// TIA Portal project "TankSimulation.TiaPortalProject" (V14)

(* hardware
DEVICE "S7-1200 station_2"  S7-1200 Station
   slot 0: "Rack_0"  S7-1200 Rack  Rack  V1.0
   slot 1: "TankSimulation"  CPU 1212C DC/DC/Rly  6ES7 212-1HE31-0XB0  V3.0
*)

// ===== PLC "TankSimulation"  CPU 1212C DC/DC/Rly =====

VAR_GLOBAL   // PLC tag table "Default tag table"
   "Tag_1" AT %M10.0 : Bool;
   "System_Byte" AT %MB1 : Byte;
   "FirstScan" AT %M1.0 : Bool;
   "DiagStatusUpdate" AT %M1.1 : Bool;
   "AlwaysTRUE" AT %M1.2 : Bool;
   "AlwaysFALSE" AT %M1.3 : Bool;
   "Clock_Byte" AT %MB0 : Byte;
   "Clock_10Hz" AT %M0.0 : Bool;
   "Clock_5Hz" AT %M0.1 : Bool;
   "Clock_2.5Hz" AT %M0.2 : Bool;
   "Clock_2Hz" AT %M0.3 : Bool;
   "Clock_1.25Hz" AT %M0.4 : Bool;
   "Clock_1Hz" AT %M0.5 : Bool;
   "Clock_0.625Hz" AT %M0.6 : Bool;
   "Clock_0.5Hz" AT %M0.7 : Bool;
END_VAR

DATA_BLOCK "Snap7interfaceDb"   // DB1
{ S7_Optimized_Access := 'FALSE' }
VERSION : 0.1
   VAR
      PumpManual : Bool;
      FlowManual : Bool;
      StartAuto : Bool;
      StopAuto : Bool;
      TankLevel : Real;
      ParameterFlowSpeed : Real := 1.0;
      ParameterPumpSpeed : Real := 2.0;
      AutoState : Bool;
      PumpsState : Bool;
      FlowState : Bool;
      RealFlowSpeed : Real;
      RealPumpSpeed : Real;
   END_VAR
BEGIN
END_DATA_BLOCK

DATA_BLOCK "StateMachineDb"   // DB2
{ S7_Optimized_Access := 'TRUE' }
VERSION : 0.1
// stored: InstanceOfName StateMachine
"StateMachine"
BEGIN
END_DATA_BLOCK

DATA_BLOCK "AlarmsDb"   // DB3
{ S7_Optimized_Access := 'FALSE' }
VERSION : 0.1
   VAR
      GlobalAlarm : Bool;
      PumpSpeedHigh : Bool;
      FlowSpeedHigh : Bool;
   END_VAR
BEGIN
END_DATA_BLOCK

FUNCTION_BLOCK "StateMachine"   // FB1, LAD
{ S7_Optimized_Access := 'TRUE' }
VERSION : 0.1
   VAR
      Clock100ms : Bool;
      "Timer" : IEC_TIMER;
      Test : Bool;
      PumpRunning : Bool;
      AutoRunning : Bool;
      FlowRunning : Bool;
      CurrentState : Byte;
   END_VAR
   VAR_TEMP   // added for the SCL form of the ladder/FBD networks
      _w1 : Bool;
   END_VAR
BEGIN

REGION Network 1: Clock 100ms
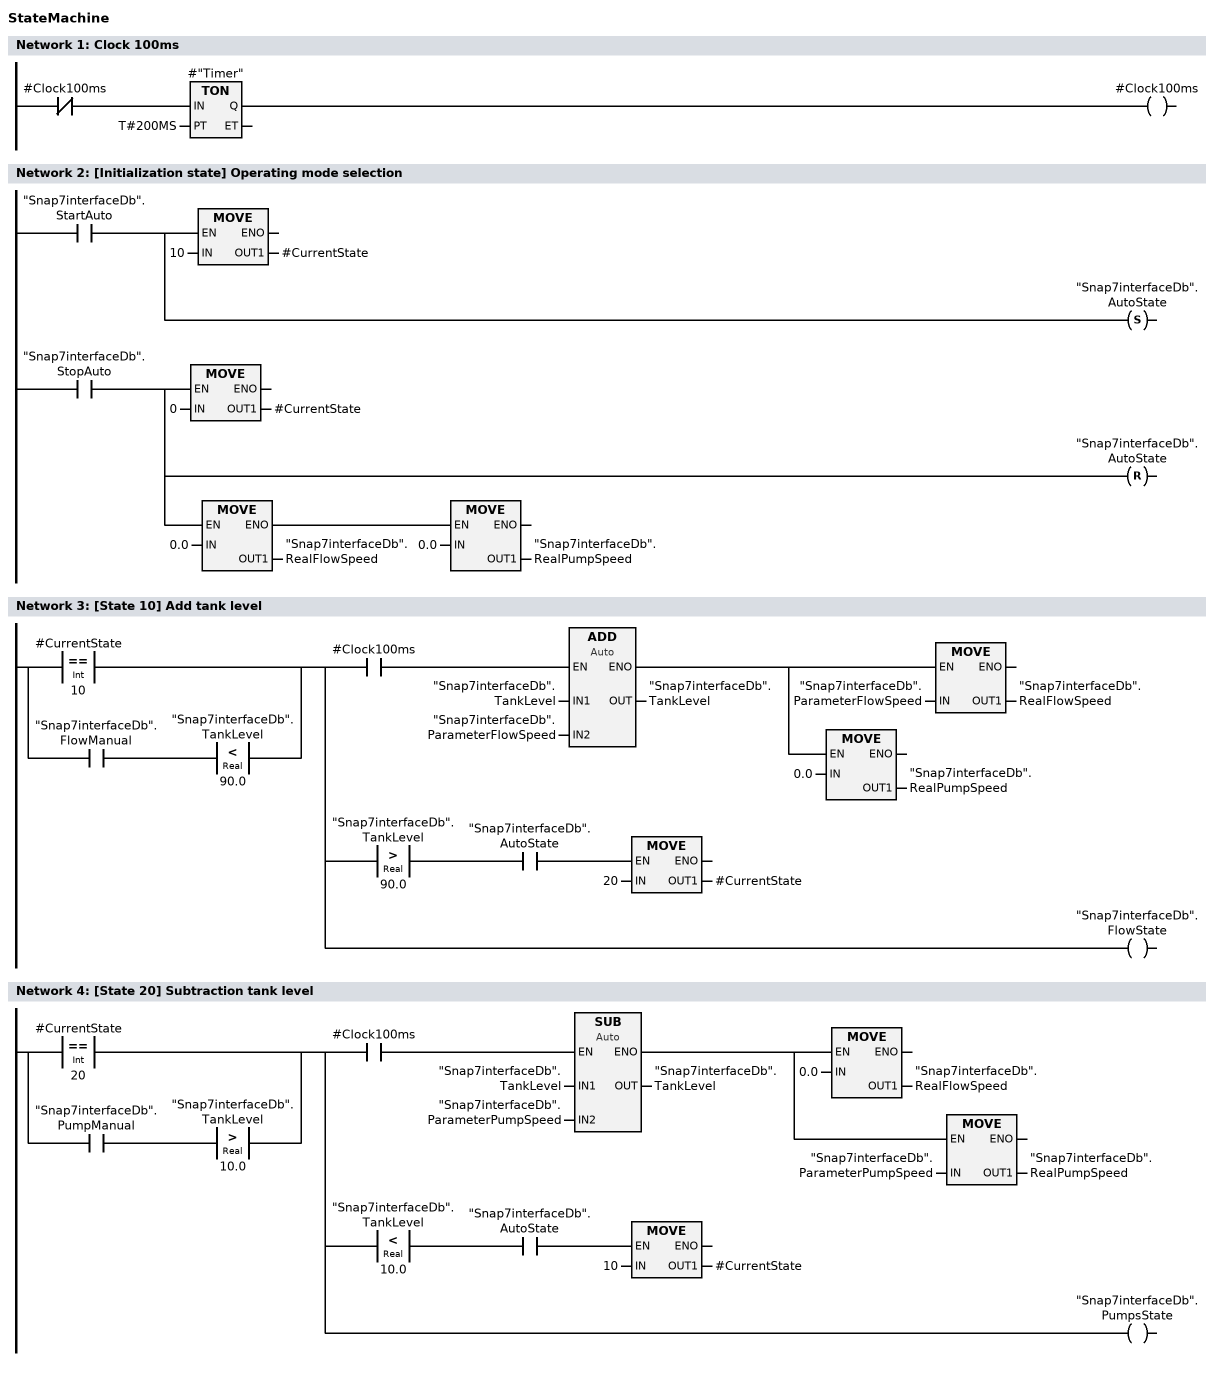
   #"Timer".TON(IN := NOT #Clock100ms, PT := T#200MS);
   #Clock100ms := #"Timer".Q;
END_REGION

REGION Network 2: [Initialization state] Operating mode selection
   RUNG wire#powerrail
      Contact( "Snap7interfaceDb".StartAuto )
      wire#w1
      { S7_GenerateENO := "TRUE" } Move(in := 10, out1 => #CurrentState)
   END_RUNG
   RUNG wire#w1
      S_Coil( "Snap7interfaceDb".AutoState )
   END_RUNG
   RUNG wire#powerrail
      Contact( "Snap7interfaceDb".StopAuto )
      wire#w2
      { S7_GenerateENO := "TRUE" } Move(in := 0, out1 => #CurrentState)
   END_RUNG
   RUNG wire#w2
      R_Coil( "Snap7interfaceDb".AutoState )
   END_RUNG
   RUNG wire#w2
      { S7_GenerateENO := "TRUE" } Move(in := 0.0, out1 => "Snap7interfaceDb".RealFlowSpeed)
      { S7_GenerateENO := "TRUE" } Move(in := 0.0, out1 => "Snap7interfaceDb".RealPumpSpeed)
   END_RUNG
   // the same network as SCL:
   // ENO of a box is taken as its EN; it also drops when the box reports an error
   IF "Snap7interfaceDb".StartAuto THEN
       #CurrentState := 10;
       "Snap7interfaceDb".AutoState := TRUE;
   END_IF;
   IF "Snap7interfaceDb".StopAuto THEN
       #CurrentState := 0;
       "Snap7interfaceDb".AutoState := FALSE;
       "Snap7interfaceDb".RealFlowSpeed := 0.0;
       "Snap7interfaceDb".RealPumpSpeed := 0.0;
   END_IF;
END_REGION

REGION Network 3: [State 10] Add tank level
   RUNG wire#powerrail
      { S7_Templates := "SrcType := Int" } EQ_Contact(in1 := #CurrentState, in2 := 10)
      wire#w1
      Contact( #Clock100ms )
      { S7_GenerateENO := "TRUE" } Add(in1 := "Snap7interfaceDb".TankLevel, in2 := "Snap7interfaceDb".ParameterFlowSpeed, out => "Snap7interfaceDb".TankLevel)
      wire#w2
      { S7_GenerateENO := "TRUE" } Move(in := "Snap7interfaceDb".ParameterFlowSpeed, out1 => "Snap7interfaceDb".RealFlowSpeed)
   END_RUNG
   RUNG wire#powerrail
      Contact( "Snap7interfaceDb".FlowManual )
      { S7_Templates := "SrcType := Real" } LT_Contact(in1 := "Snap7interfaceDb".TankLevel, in2 := 90.0)
   END_RUNG wire#w1
   RUNG wire#w2
      { S7_GenerateENO := "TRUE" } Move(in := 0.0, out1 => "Snap7interfaceDb".RealPumpSpeed)
   END_RUNG
   RUNG wire#w1
      { S7_Templates := "SrcType := Real" } GT_Contact(in1 := "Snap7interfaceDb".TankLevel, in2 := 90.0)
      Contact( "Snap7interfaceDb".AutoState )
      { S7_GenerateENO := "TRUE" } Move(in := 20, out1 => #CurrentState)
   END_RUNG
   RUNG wire#w1
      Coil( "Snap7interfaceDb".FlowState )
   END_RUNG
   // the same network as SCL:
   // ENO of a box is taken as its EN; it also drops when the box reports an error
   #_w1 := (#CurrentState = 10) OR ("Snap7interfaceDb".FlowManual AND ("Snap7interfaceDb".TankLevel < 90.0));
   IF #_w1 AND #Clock100ms THEN
       "Snap7interfaceDb".TankLevel := "Snap7interfaceDb".TankLevel + "Snap7interfaceDb".ParameterFlowSpeed;
       "Snap7interfaceDb".RealFlowSpeed := "Snap7interfaceDb".ParameterFlowSpeed;
       "Snap7interfaceDb".RealPumpSpeed := 0.0;
   END_IF;
   IF #_w1 AND ("Snap7interfaceDb".TankLevel > 90.0) AND "Snap7interfaceDb".AutoState THEN
       #CurrentState := 20;
   END_IF;
   "Snap7interfaceDb".FlowState := #_w1;
END_REGION

REGION Network 4: [State 20] Subtraction tank level
   RUNG wire#powerrail
      { S7_Templates := "SrcType := Int" } EQ_Contact(in1 := #CurrentState, in2 := 20)
      wire#w1
      Contact( #Clock100ms )
      { S7_GenerateENO := "TRUE" } Sub(in1 := "Snap7interfaceDb".TankLevel, in2 := "Snap7interfaceDb".ParameterPumpSpeed, out => "Snap7interfaceDb".TankLevel)
      wire#w2
      { S7_GenerateENO := "TRUE" } Move(in := 0.0, out1 => "Snap7interfaceDb".RealFlowSpeed)
   END_RUNG
   RUNG wire#powerrail
      Contact( "Snap7interfaceDb".PumpManual )
      { S7_Templates := "SrcType := Real" } GT_Contact(in1 := "Snap7interfaceDb".TankLevel, in2 := 10.0)
   END_RUNG wire#w1
   RUNG wire#w2
      { S7_GenerateENO := "TRUE" } Move(in := "Snap7interfaceDb".ParameterPumpSpeed, out1 => "Snap7interfaceDb".RealPumpSpeed)
   END_RUNG
   RUNG wire#w1
      { S7_Templates := "SrcType := Real" } LT_Contact(in1 := "Snap7interfaceDb".TankLevel, in2 := 10.0)
      Contact( "Snap7interfaceDb".AutoState )
      { S7_GenerateENO := "TRUE" } Move(in := 10, out1 => #CurrentState)
   END_RUNG
   RUNG wire#w1
      Coil( "Snap7interfaceDb".PumpsState )
   END_RUNG
   // the same network as SCL:
   // ENO of a box is taken as its EN; it also drops when the box reports an error
   #_w1 := (#CurrentState = 20) OR ("Snap7interfaceDb".PumpManual AND ("Snap7interfaceDb".TankLevel > 10.0));
   IF #_w1 AND #Clock100ms THEN
       "Snap7interfaceDb".TankLevel := "Snap7interfaceDb".TankLevel - "Snap7interfaceDb".ParameterPumpSpeed;
       "Snap7interfaceDb".RealFlowSpeed := 0.0;
       "Snap7interfaceDb".RealPumpSpeed := "Snap7interfaceDb".ParameterPumpSpeed;
   END_IF;
   IF #_w1 AND ("Snap7interfaceDb".TankLevel < 10.0) AND "Snap7interfaceDb".AutoState THEN
       #CurrentState := 10;
   END_IF;
   "Snap7interfaceDb".PumpsState := #_w1;
END_REGION
END_FUNCTION_BLOCK

FUNCTION "Alarms" : Void   // FC1, LAD
{ S7_Optimized_Access := 'TRUE' }
VERSION : 0.1
BEGIN

REGION Network 1: DB3.DBX0.2 - [Alarm] Flow speed high
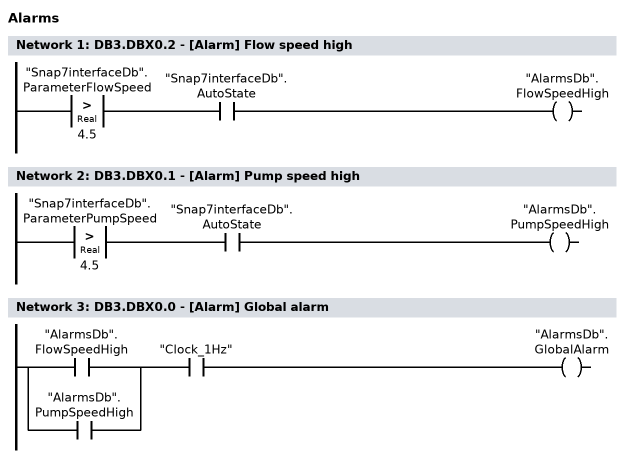
   RUNG wire#powerrail
      { S7_Templates := "SrcType := Real" } GT_Contact(in1 := "Snap7interfaceDb".ParameterFlowSpeed, in2 := 4.5)
      Contact( "Snap7interfaceDb".AutoState )
      Coil( "AlarmsDb".FlowSpeedHigh )
   END_RUNG
   // the same network as SCL:
   "AlarmsDb".FlowSpeedHigh := ("Snap7interfaceDb".ParameterFlowSpeed > 4.5) AND "Snap7interfaceDb".AutoState;
END_REGION

REGION Network 2: DB3.DBX0.1 - [Alarm] Pump speed high
   RUNG wire#powerrail
      { S7_Templates := "SrcType := Real" } GT_Contact(in1 := "Snap7interfaceDb".ParameterPumpSpeed, in2 := 4.5)
      Contact( "Snap7interfaceDb".AutoState )
      Coil( "AlarmsDb".PumpSpeedHigh )
   END_RUNG
   // the same network as SCL:
   "AlarmsDb".PumpSpeedHigh := ("Snap7interfaceDb".ParameterPumpSpeed > 4.5) AND "Snap7interfaceDb".AutoState;
END_REGION

REGION Network 3: DB3.DBX0.0 - [Alarm] Global alarm
   RUNG wire#powerrail
      Contact( "AlarmsDb".FlowSpeedHigh )
      wire#w1
      Contact( "Clock_1Hz" )
      Coil( "AlarmsDb".GlobalAlarm )
   END_RUNG
   RUNG wire#powerrail
      Contact( "AlarmsDb".PumpSpeedHigh )
   END_RUNG wire#w1
   // the same network as SCL:
   "AlarmsDb".GlobalAlarm := ("AlarmsDb".FlowSpeedHigh OR "AlarmsDb".PumpSpeedHigh) AND "Clock_1Hz";
END_REGION
END_FUNCTION

ORGANIZATION_BLOCK "Main"   // OB1, LAD, ProgramCycle
TITLE = "Main Program Sweep (Cycle)"
{ S7_Optimized_Access := 'TRUE' }
VERSION : 0.1
   VAR_INPUT
      Initial_Call : Bool;   // Initial call of this OB
      Remanence : Bool;   // =True, if remanent data are available
   END_VAR
BEGIN

REGION Network 1
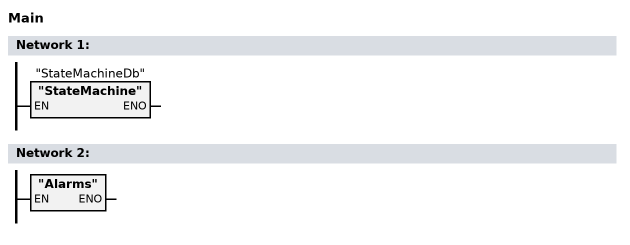
   RUNG wire#powerrail
      "StateMachineDb"()
   END_RUNG
   // the same network as SCL:
   "StateMachineDb"();   // "StateMachine"
END_REGION

REGION Network 2
   RUNG wire#powerrail
      "Alarms"()
   END_RUNG
   // the same network as SCL:
   "Alarms"();
END_REGION
END_ORGANIZATION_BLOCK